// TIA Portal V16 export
// export: Created 2024-04-26T21:24:43.9818457Z, ExportSetting WithDefaults, DisplayName Totally Integrated Automation Portal, DisplayVersion V16, DisplayName TIA Portal Version Control Interface, DisplayVersion V16, DisplayName TIA Portal Openness, DisplayVersion V16, DisplayName STEP 7 Professional, DisplayVersion V16, DisplayName STEP 7 Safety, DisplayVersion V16, DisplayName WinCC Professional, DisplayVersion V16
DATA_BLOCK "MC_MoveAbsolute_DB_2"   // DB27
// stored: AutoNumber true, InstanceOfName MC_MoveAbsolute, OfSystemLibElement MC_MoveAbsolute, OfSystemLibVersion 6.0
"MC_MoveAbsolute"
   // VAR_INPUT
   //    Axis : TO_PositioningAxis;
   //    Execute : Bool;
   //    Position : Real;
   //    Velocity : Real;
   //    Direction : Int;
   // END_VAR
   // VAR_OUTPUT
   //    Done : Bool;
   //    Busy : Bool;
   //    CommandAborted : Bool;
   //    Error : Bool;
   //    ErrorID : Word;
   //    ErrorInfo : Word;
   // END_VAR
   // VAR
   //    FB_ID : DInt;
   // END_VAR
BEGIN
END_DATA_BLOCK
